FUNCTION derivcvar_M_HardwareMap_t : LREAL
VAR_INPUT
	state: STATE;
END_VAR

derivcvar_M_HardwareMap_t := 1.0;

END_FUNCTION

(* stored: Version 1.1.0.1, ProductVersion 3.1.4022.18
   POU derivcvar_M_HardwareMap_t: Id {68d39212-cbf0-4230-b034-2ebb3f9b66ba}, SpecialFunc None *)
